PROGRAM MAIN
VAR
	bStateC			AT%I*		: BOOL;
	bStateH			AT%I*		: BOOL;
	byStateH_C					: BYTE;				//{#lynus.ag#()}
	byErrorWarning				: BYTE;				//{#lynus.ag#()}
	byReady						: BYTE;				//{#lynus.ag#()}
	byHB						: BYTE;				//{#lynus.ag#()}
	rHKBKA_RT1	 	AT%I*		: LREAL;			//{#lynus.ag#()}
	rHKBKA_RT2	 	AT%I*		: LREAL;			//{#lynus.ag#()}
	rHKBKA_RT3	 	AT%I*		: LREAL;			//{#lynus.ag#()}
	rHKBKA_FlowT	AT%I*		: LREAL;			//{#lynus.ag#()}
	rNewFlowTemp				: LREAL;			//{#lynus.ag#()}
END_VAR

//State for Heatin gor Cooling
byStateH_C := 0;
	IF bStateC THEN byStateH_C := 2; END_IF
		IF bStateH THEN byStateH_C := 1; END_IF

END_PROGRAM

(* stored: Version 1.1.0.1, ProductVersion 3.1.4024.9
   POU MAIN: Id {eea8685a-b6e3-453b-8588-b15818aca6ba}, SpecialFunc None *)
